FUNCTION_BLOCK T_GetComponentIndexOutOfBoundaryResultsFalse EXTENDS T_UnitTestBase
VAR
  list : T_ComponentsCollection;
  newComponent : T_ComponentMock;
  actual : I_ComponentBase;
  expected : I_ComponentBase;
  result, tryGetResultWithinMax, tryGetResultAboveMax : BOOL;
END_VAR

list.AddComponent(newComponent);

tryGetResultWithinMax := NOT list.TryGetComponent(3, component => actual);
tryGetResultAboveMax := NOT list.TryGetComponent(13, component => actual);

result := actual = 0;
assertion.AssertEquals_BOOL(TRUE, result, 'result');
assertion.AssertEquals_BOOL(TRUE, tryGetResultWithinMax, 'tryGetResultWithinMax');
assertion.AssertEquals_BOOL(TRUE, tryGetResultAboveMax, 'tryGetResultAboveMax');
TestFinished();

END_FUNCTION_BLOCK

(* stored: Version 1.1.0.1, ProductVersion 3.1.4024.12
   POU T_GetComponentIndexOutOfBoundaryResultsFalse: Id {f7c8f7ba-ae31-41e2-85cc-10eb490f1c48}, SpecialFunc None *)
